TYPE MaterialBlock EXTENDS MaterialHeader :
STRUCT
	data : ARRAY[1..112] of WORD;
END_STRUCT
END_TYPE

(* stored: Version 1.1.0.1, ProductVersion 3.1.4020.12
   DUT MaterialBlock: Id {8bc725df-9215-4403-8bfc-761ebea6ca5e} *)
